Universal Robots URScript: test_modified.script

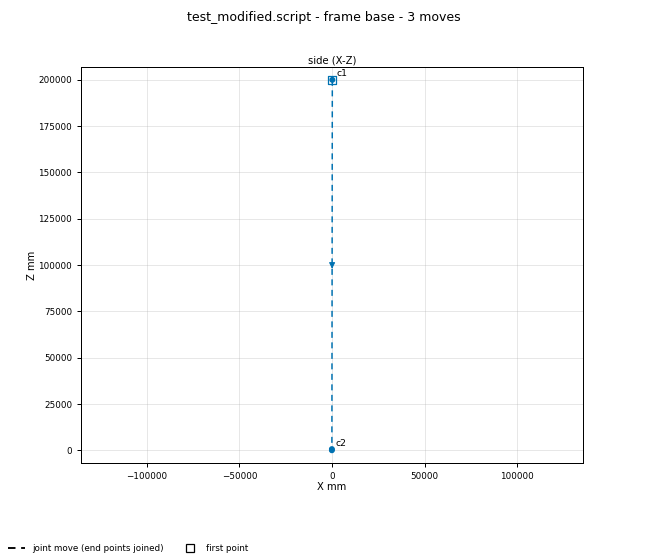
[picture p0: tool path of test_modified.script in frame base, 3 of 3 moves have a stored position in this frame; points joined in program order, loops and branches not executed]
def Test():
  global _hidden_verificationVariable=0
  step_count_0ff553c9_31d9_4e1b_936b_c32f9b27ad0c = 0.0
  thread Step_Counter_Thread_99b7fb34_fe38_4c53_a84f_0ec64a1a24ca():
    while (True):
      step_count_0ff553c9_31d9_4e1b_936b_c32f9b27ad0c = step_count_0ff553c9_31d9_4e1b_936b_c32f9b27ad0c + 1.0
      sync()
    end
  end
  run Step_Counter_Thread_99b7fb34_fe38_4c53_a84f_0ec64a1a24ca()
  set_tool_communication(False, 115200, 0, 1, 1.5, 3.5)
  set_tool_output_mode(0)
  set_tool_digital_output_mode(0, 1)
  set_tool_digital_output_mode(1, 1)
  set_tool_voltage(0)
  set_gravity([0.0, 0.0, 9.82])
  set_standard_analog_input_domain(0, 1)
  set_standard_analog_input_domain(1, 1)
  set_tool_analog_input_domain(0, 1)
  set_tool_analog_input_domain(1, 1)
  set_analog_outputdomain(0, 0)
  set_analog_outputdomain(1, 0)
  set_input_actions_to_default()
  set_safety_mode_transition_hardness(1)
  set_tcp(p[0.0,0.0,0.11,0.0,0.0,0.0])
  set_target_payload(0.530000, [0.009000, -0.039000, 0.092000], [0.000534, 0.000534, 0.000534, 0.000000, 0.000000, 0.000000])
  global Al_plate=p[0.12405209206180495,-0.2666666051843552,0.020008101224669964,-9.276623980477388E-5,1.8107917580596192E-5,3.1233857134705927]
  global Frame2x2=p[0.18266245434305164,-0.34273121659514855,0.026002571110600767,-2.225423529876215E-4,3.0110667546023537E-4,3.1233976058306383]
  global URlogoTutorial=p[-0.08178353973148575,-0.3363174165299142,0.04788621506469384,-3.9746155723688456E-5,-3.4682148779121894E-5,-1.5668291789091222]
  global carouselrod=p[0.2020731702281844,-0.34951442511341274,0.1947611446273096,3.139766958234101,-0.10689428010274801,-1.1796370330365635E-5]
  global paper=p[-0.09670794781244417,-0.3283412964648025,0.027665994240809913,-3.2057893450593004E-5,2.867088716161181E-5,-1.6085327915291054]
  global rod=p[0.13368013097420872,-0.41123185103490206,0.09926814901395645,2.2214229924093103,-2.2214158162465862,-2.9165882738638143E-5]
  # begin: URCap Installation Node
  #   Source: External Control, 1.0.5, FZI Research Center for Information Technology
  #   Type: External Control
  # end: URCap Installation Node
  global c1_p=p[0.11122465956611277, -0.1651270323018603, 200.0, 0, 3.14159, 0]
  global c1_q=[1.4769117051943825, -1.8610464984796677, 1.8741644486163223, -1.583914276931551, -1.5707963267948966, 1.4769117051943825]
  global c2_p=p[-.125097928533, -.379144222044, .070861676824, -3.139810722682, .105446315316, .000070958941]
  global c2_q=[-1.5585409219037167, -2.0100444173139564, -1.6214680589971655, -1.0785837695635507, 1.5737966620464547, 3.2257491810537076]
  global Waypoint_1_p=p[-.127484884293, -.225752120702, .684570412903, 1.614441233679, -.056082236805, .077311990652]
  global Waypoint_1_q=[-1.5585258642788755, -1.6125626661427257, 0.0, -1.5707963267948966, 1.5737857818617464, 3.2257497310681664]
  while (True):
    $ 2 "Robot Program"
    $ 3 "MoveJ"
    $ 4 "c1" "breakAfter"
    movej(get_inverse_kin(c1_p, qnear=c1_q), a=0.5, v=1)
    $ 5 "Wait: 5.0"
    sleep(5.0)
    $ 6 "c2" "breakAfter"
    movej(get_inverse_kin(c2_p, qnear=c2_q), a=0.5, v=1)
    $ 7 "Wait: 5.0"
    sleep(5.0)
    $ 8 "Waypoint_1" "breakAfter"
    movej(get_inverse_kin(Waypoint_1_p, qnear=Waypoint_1_q), a=0.5, v=1)
    $ 9 "Wait: 2.0"
    sleep(2.0)
  end
end
